TYPE E_SYSTEM_MaintainFolders :
(
	E_FOLDER_IDLE,
	E_FOLDER_ININT_CHECK,
	E_FOLDER_CHECK,
	E_FOLDER_CREATEBASEPATH,
	E_FOLDER_DELETE,
	E_FOLDER_DONE
);
END_TYPE

(* stored: Version 1.1.0.1
   DUT E_SYSTEM_MaintainFolders: Id {7c7a7ba4-7cdc-4901-a9ce-08be52977c96} *)
